{attribute 'GeneratedUsingTerminal: ER7041-0002-0024'}
{attribute addProperty BoxType "ER7041-0002-0024"}
{attribute addProperty Id "StatusAT %I*Status_B679584511"}
{attribute addProperty CRC "921504111"}
{attribute addProperty Size "11"}
TYPE STM_Status_36ED096F EXTENDS InputBase_8311D824 :
STRUCT
	{attribute addProperty Name "Status"}
	Status AT %I* : Status_B6795845;
END_STRUCT
END_TYPE

(* stored: Version 1.2.0.0, ProductVersion 3.1.4024.11
   DUT STM_Status_36ED096F: Id {adfdf1d6-0a51-4bea-a448-a83bff3829eb} *)
